TYPE ST_Control :
STRUCT
	
	ManualMode : BOOL;

END_STRUCT
END_TYPE

(* stored: Version 1.1.0.1, ProductVersion 3.1.4024.12
   DUT ST_Control: Id {3c5f0bae-9e6c-40dc-8529-3bd5edaff156} *)
